TYPE Vec13di : ARRAY[1..13] OF DINT; END_TYPE

(* stored: Version 1.1.0.1, ProductVersion 3.1.4024.12
   DUT Vec13di: Id {df0b9a7a-8e0c-4f17-9aa5-4a8ce6ecb5e5} *)
